TYPE ST_Event :
STRUCT
END_STRUCT
END_TYPE

(* stored: Version 1.1.0.1, ProductVersion 3.1.4024.12
   DUT ST_Event: Id {33a87115-0f2f-4a04-9f80-e5673a0dd10f} *)
